// TwinCAT 3 PLC project P1
// ProgramVersion: 3.1.4024.0
// libraries:
//   Tc2_Standard, * (Beckhoff Automation GmbH)
//   Tc2_System, * (Beckhoff Automation GmbH)
//   Tc3_Module, * (Beckhoff Automation GmbH)
// project tree:
//   / PlcTask.TcTTO
//   POUs/ MAIN.TcPOU
// real-time tasks:
//   TASK PlcTask: cycle T#10ms, priority 20, ADS port 350

CONFIGURATION P1
    RESOURCE PLC ON TwinCAT3
        TASK PlcTask(INTERVAL := T#10ms, PRIORITY := 20);
        PROGRAM MAIN WITH PlcTask : MAIN;
    END_RESOURCE
END_CONFIGURATION

// ---- POUs/MAIN.TcPOU
PROGRAM MAIN
VAR
	stop: BOOL;
	start: BOOL;
	R1: BOOL;
	R2: BOOL;
	weight: INT;
	binASorter: BOOL;
	binBSorter: BOOL;
END_VAR

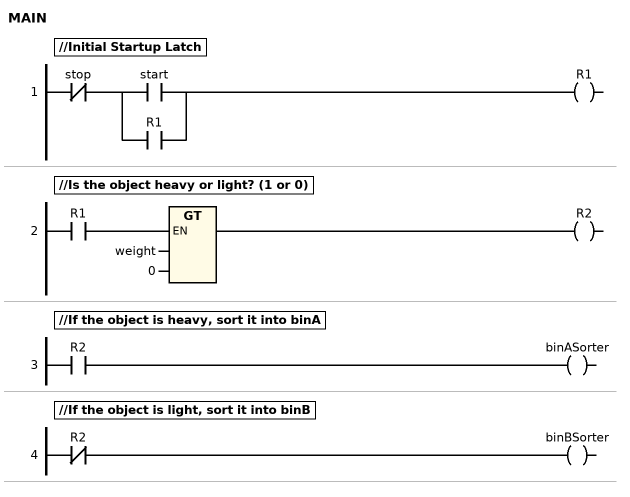
// NETWORK 1
// label: //Initial Startup Latch
R1 := NOT stop AND (start OR R1);

// NETWORK 2
// label: //Is the object heavy or light? (1 or 0)
R2 := R1 AND weight > 0;

// NETWORK 3
// label: //If the object is heavy, sort it into binA
binASorter := R2;

// NETWORK 4
// label: //If the object is light, sort it into binB
binBSorter := NOT R2;

END_PROGRAM
